Universal Robots PolyScope program: if_96.urp

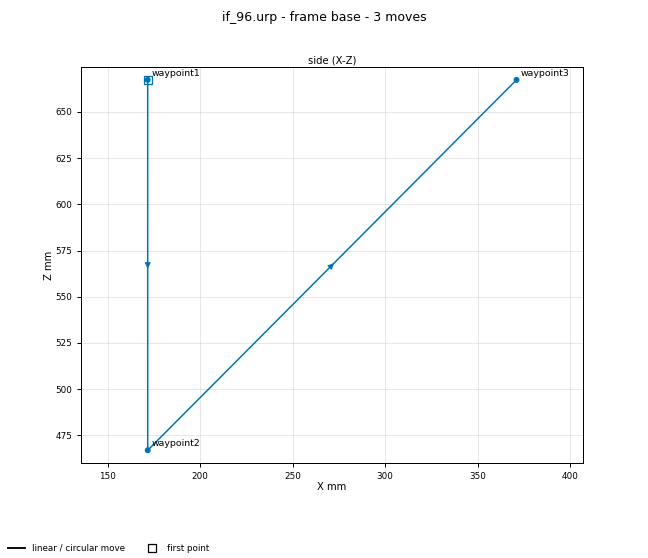
[picture p0: tool path of if_96.urp in frame base, 3 of 3 moves have a stored position in this frame; points joined in program order, loops and branches not executed]
Program if_96 (createdIn=3.2.19293 lastSavedIn=3.2.19293 directory=/programs installation=default robotSerialNumber=2015351391)
Calibrated DH parameters: a=[0.000352, -0.161198, -0.373486, 0.00005, 0.000049, 0]; d=[0.089268, 352.477598, -320.08558, -32.281492, 0.094939, 0.082518]; alpha=[1.570728, 0.001116, -0.003686, 1.571189, -1.570572, 0]; deltaTheta=[-0.000012, 1.181849, -1.491165, 0.309495, -0.000007, 0.000025]
Robot Program (runOnlyOnce=false motionType=MoveJ speed=1.047198 acceleration=1.396263 recalculateMotions=false)
  MoveL speed 250 mm/s, acceleration 1200 mm/s^2 (recalculateMotions=false) feature=Base
    Waypoint waypoint1: TCP in base x=171.583 y=236.698 z=667.293 mm, rx=-1.5849 ry=-0.1094 rz=-0.2822 rad; joints [73.416, -64.137, -100.793, -15.776, 100.192, -14.656] deg
    If Button≟ True (checkContinuously=true)
      Waypoint waypoint2: TCP in base x=171.6 y=236.701 z=466.995 mm, rx=-1.585 ry=-0.1092 rz=-0.2824 rad; joints [73.34, -64.034, -130.449, 13.786, 100.363, -14.629] deg
    Else 
      Waypoint waypoint3: TCP in base x=371.022 y=236.741 z=667.271 mm, rx=-1.585 ry=-0.1093 rz=-0.2823 rad; joints [39.628, -88.343, -82.922, -9.865, 134.019, -15.246] deg
